Staubli VAL3: pick_cells.pgx

program pick_cells(num x_nNum_choose)
  local num l_nNum_cRow
  local num l_nNum_cCol
  local point l_pPoint_cur
  local tool l_tTool_cur
  local point l_pPoint_lb_cur
  local num l_nNum_total
  local num l_nNum_current
  local dio l_dDio_cur_cy
  local dio l_dDio_secure
begin
  //pick from f1 put to bin
  call show_check("Reload")

  switch x_nNum_choose
    case 1
      //f1
      l_tTool_cur = t1
      dioLink(l_dDio_cur_cy,dDio_t1_cy)
      dioLink(l_dDio_secure,dDio_f1_secure)
      //dio assignment
    break
    case 2
      //f2
      l_tTool_cur = t2
      dioLink(l_dDio_cur_cy,dDio_t2_cy)
      dioLink(l_dDio_secure,dDio_f2_secure)
      //dio assignment
    break
    case 3
      //f3
      l_tTool_cur = t3
      dioLink(l_dDio_cur_cy,dDio_t3_cy)
      dioLink(l_dDio_secure,dDio_f3_secure)
      //dio assignment
    break

  endSwitch

  //calculate total
  call calculate_total(x_nNum_choose,l_nNum_total)

  for l_nNum_current=0 to(l_nNum_total-1) step 1

    //show progress
    call show_progress(sScreen_ppShelf,l_nNum_current+1,l_nNum_total,6)

    //row,col count
    call calculate_rc(l_nNum_current,x_nNum_choose,l_nNum_cRow,l_nNum_cCol)
    //pick position count
    call calculate_pick(l_nNum_cRow,l_nNum_cCol,l_pPoint_cur,x_nNum_choose)
    //pick (not defined yet
    call regular_pick(l_tTool_cur,mNomSpeed,mSlowSpeed,l_pPoint_cur,l_dDio_cur_cy,false,l_dDio_secure)

    //bin place (bin not defined yet
    call regular_place(l_tTool_cur,mNomSpeed,mSlowSpeed,ref,false,l_dDio_cur_cy,false)

  endFor

end
